TYPE "AGV_ShW"
VERSION : 0.1
   STRUCT
      Trigger : Bool;
      Result : Int;
      Completed : Bool;
      TaskNo : Int;
      PointName : String[48];
      materialLot : String[48];
      materialQuantity : Int;
      SafetySignal : Bool;
      ProcessBit : Bool;
   END_STRUCT;

END_TYPE

